SUBAPPLICATION Select_EnableOk_AX (* Wie MyLib::sys::Select_EnableOk, aber vollstaendig adapter-nativ: bEnable/bOk kommen als AX-Adapter, value geht als AUS-Adapter raus - kein Event-Handling noetig, jede Aenderung an bEnable/bOk propagiert automatisch ueber die Adapter-Kette. *)
  (* Standard: 61499-2; Description: Copyright (c) 2026 Meisterschulen am Ostbahnhof This program and the accompanying materials are made available under the terms of the Eclipse Public License 2.0 which is available at https://www.eclipse.org/legal/epl-2.0/ SPDX-License-Identifier: EPL-2.0 *)
  (* Version 1.1, 2026-08-31, Franz Höpfinger, Meisterschulen am Ostbahnhof, Adapter-native Variante von Select_EnableOk: AUS_AX_SEL_AUS (2-stufig) statt F_SEL+Event-Merge, initval_AUS speist die 3 Parameter-Werte als Adapter ein - kein REQ/CNF mehr auf dieser Ebene *)
  PACKAGE MyLib::sys;
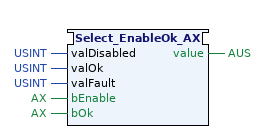
  VAR_INPUT
    valDisabled : USINT; (* Ausgabewert wenn bEnable=FALSE - einmalig bei Instanziierung per Parameter gesetzt *)
    valOk : USINT; (* Ausgabewert wenn bEnable=TRUE und bOk=TRUE - einmalig bei Instanziierung per Parameter gesetzt *)
    valFault : USINT; (* Ausgabewert wenn bEnable=TRUE und bOk=FALSE - einmalig bei Instanziierung per Parameter gesetzt *)
  END_VAR
  SOCKETS
    bEnable : adapter::types::unidirectional::AX; (* Aktiviert (BOOL, ueber Adapter statt Klartext) *)
    bOk : adapter::types::unidirectional::AX; (* OK-Zustand (BOOL, ueber Adapter statt Klartext) - nur relevant wenn bEnable=TRUE *)
  END_SOCKETS
  PLUGS
    value : adapter::types::unidirectional::AUS; (* Ausgewaehlter Wert *)
  END_PLUGS
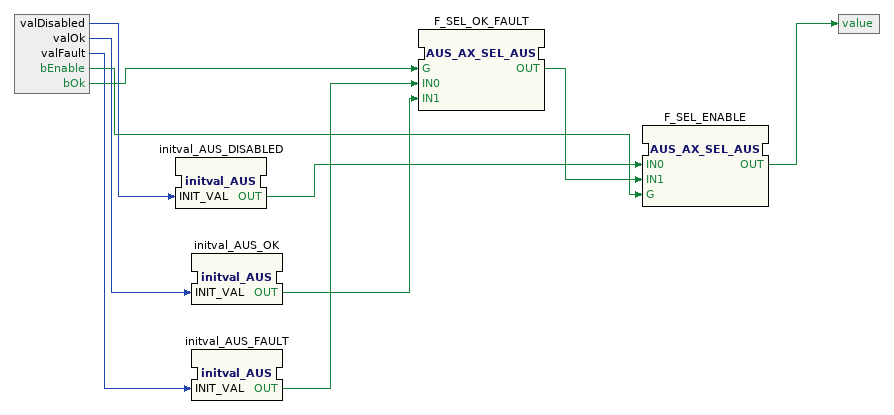
  FBS
    initval_AUS_FAULT : adapter::types::unidirectional::AUS::initval::initval_AUS;
    initval_AUS_OK : adapter::types::unidirectional::AUS::initval::initval_AUS;
    initval_AUS_DISABLED : adapter::types::unidirectional::AUS::initval::initval_AUS;
    F_SEL_OK_FAULT : adapter::iec61131::selection::AUS_AX_SEL_AUS;
    F_SEL_ENABLE : adapter::iec61131::selection::AUS_AX_SEL_AUS;
  END_FBS
  DATA_CONNECTIONS
    valFault TO initval_AUS_FAULT.INIT_VAL;
    valOk TO initval_AUS_OK.INIT_VAL;
    valDisabled TO initval_AUS_DISABLED.INIT_VAL;
  END_CONNECTIONS
  ADAPTER_CONNECTIONS
    bOk TO F_SEL_OK_FAULT.G;
    initval_AUS_FAULT.OUT TO F_SEL_OK_FAULT.IN0;
    initval_AUS_OK.OUT TO F_SEL_OK_FAULT.IN1;
    initval_AUS_DISABLED.OUT TO F_SEL_ENABLE.IN0;
    F_SEL_OK_FAULT.OUT TO F_SEL_ENABLE.IN1;
    bEnable TO F_SEL_ENABLE.G;
    F_SEL_ENABLE.OUT TO value;
  END_CONNECTIONS
END_SUBAPPLICATION
